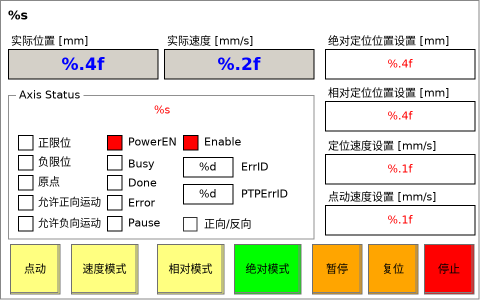
VISUALIZATION motionModuleP1  // 480x300
VAR_IN_OUT
	userData: motionModuleDataHMI;	
END_VAR
    Button (10,244 50x50), "点动", input disabled if: NOT userData.jogCondition OR NOT userData.ctrlModeCondition
        tap userData.manJogGo
    Button (157,244 67x50), "相对模式", tooltip "Please keep pressing to trigger", input disabled if: NOT userData.relCondition OR NOT userData.ctrlModeCondition
        tap userData.manRelGo
    Button (234,244 67x50), "绝对模式", tooltip "Please keep pressing to trigger", input disabled if: NOT userData.absCondition OR NOT userData.ctrlModeCondition
        tap userData.manABSGo
    Button (424,244 50x50), "停止"
        tap userData.stop
    Rectangle (8,49 150x30), "%.4f", text variable: userData.actualPos
    Rectangle (8,26 150x30), "实际位置 [mm]"
    Rectangle (164,49 150x30), "%.2f", text variable: userData.actualVel
    Rectangle (164,26 150x30), "实际速度 [mm/s]"
    Rectangle (325,79 145x28), "相对定位位置设置 [mm]"
    Rectangle (325,26 150x30), "绝对定位位置设置 [mm]"
    Rectangle (325,131 150x30), "定位速度设置 [mm/s]"
    GroupBox (8,87 306x152), "Axis Status"
        Rectangle (99,48 15x15), colour toggle: userData.powerEnable
        Rectangle (117,44 64x22), "PowerEN"
        Rectangle (10,48 15x15), colour toggle: userData.forwardLimitSwitch
        Rectangle (10,68 15x15), colour toggle: userData.backwardsLimitSwitch
        Rectangle (10,88 15x15), colour toggle: userData.dogPointSwitch
        Rectangle (27,84 64x22), "原点"
        Rectangle (99,68 15x15), colour toggle: userData.busy
        Rectangle (117,66 64x22), "Busy"
        Rectangle (230,69 46x22), "ErrID"
        Rectangle (27,104 67x22), "允许正向运动"
        Rectangle (10,108 15x15), colour toggle: userData.forwardEnable
        Rectangle (27,125 67x22), "允许负向运动"
        Rectangle (10,129 15x15), colour toggle: userData.backwardsEnable
        Rectangle (117,85 64x22), "Done"
        Rectangle (117,105 64x22), "Error"
        Rectangle (175,97 50x20), "%d", text variable: userData.PTPErrID
        Rectangle (99,129 15x15), colour toggle: userData.oPause
        Rectangle (117,125 64x22), "Pause"
        Rectangle (27,45 68x22), "正限位"
        Rectangle (27,64 64x22), "负限位"
        Rectangle (175,70 50x20), "%d", text variable: userData.errID
        Rectangle (175,48 15x15), colour toggle: userData.enable
        Rectangle (230,96 64x22), "PTPErrID"
        Rectangle (99,88 15x15), colour toggle: userData.done
        Rectangle (99,108 15x15), colour toggle: userData.error
        Checkbox (173,122 130x30), "正向/反向", variable: userData.choiceOfDirection
        Rectangle (193,44 52x22), "Enable"
    Rectangle (12,100 300x20), "%s", text variable: userData.errTxt
    Rectangle (325,49 150x30), "%.4f", text variable: userData.manABSPos, input disabled if: Not userData.goHomeDone
        OnMouseDown: write the text variable via Edit
    Rectangle (325,101 150x30), "%.4f", text variable: userData.manRelDis
        OnMouseDown: write the text variable via Edit
    Rectangle (325,154 150x30), "%.1f", text variable: userData.manVel
        OnMouseDown: write the text variable via Edit
    Rectangle (325,182 150x30), "点动速度设置 [mm/s]"
    Rectangle (325,205 150x30), "%.1f", text variable: userData.manJogVel
        OnMouseDown: write the text variable via Edit
    Button (71,244 67x50), "速度模式", invisible if: FALSE, input disabled if: NOT userData.velCondition OR NOT userData.ctrlModeCondition
        tap userData.manVelGo
    Button (368,244 50x50), "复位"
        tap userData.reset
    Rectangle (5,5 467x20), "%s", text variable: userData.nameTXT
    Button (312,244 50x50), "暂停", colour toggle: userData.oPause, input disabled if: NOT userData.ctrlModeCondition
        tap userData.pauseB
END_VISUALIZATION

(* stored: Version 1.1.0.1, ProductVersion 3.1.4024.4
   Visu motionModuleP1: Id {322c88a5-6a1b-4fff-895c-11a53f03b04c} *)
